// TwinCAT 3 PLC project plc_project
// ProgramVersion: 3.1.4022.1
// libraries:
//   Tc2_Standard, * (Beckhoff Automation GmbH)
//   Tc2_System, * (Beckhoff Automation GmbH)
//   Tc3_Module, * (Beckhoff Automation GmbH)
//   VisuDialogs, * (System)
//   VisuSymbols,3.5.10.0,System
// project tree:
//   / GlobalTextList.TcGTLO, PlcTask.TcTTO, Visualization Manager.TcVMO (not stored)
//   POUs/ MAIN.TcPOU, POU.TcPOU
//   VISUs/ Visualization.TcVIS

CONFIGURATION plc_project
    RESOURCE PLC ON TwinCAT3
        TASK PlcTask(INTERVAL := T#10ms, PRIORITY := 20);
        PROGRAM MAIN WITH PlcTask : MAIN;
    END_RESOURCE
END_CONFIGURATION

// ---- POUs/MAIN.TcPOU
PROGRAM MAIN
VAR
END_VAR

POU();

END_PROGRAM

// ---- POUs/POU.TcPOU
PROGRAM POU
VAR
	A: BOOL;
	B: BOOL;
	C: BOOL:= FALSE;
	add_result: UINT;
	sub_result: INT;
	mul_result: REAL;
	div_result: REAL;
	TON_0: TON;
	ton0_et: TIME;
	TOF_0: TOF;
	tof0_et: TIME;
	TP_0: TP;
	tp0_et: TIME;
	D: BOOL;
	CTD_0: CTD;
	CTD_1: CTD;
	ctd1_cv: WORD;
	Zero: BOOL;
	CTU_0: CTU;
	ctu0_cv: WORD;
	Maximum: BOOL;
END_VAR

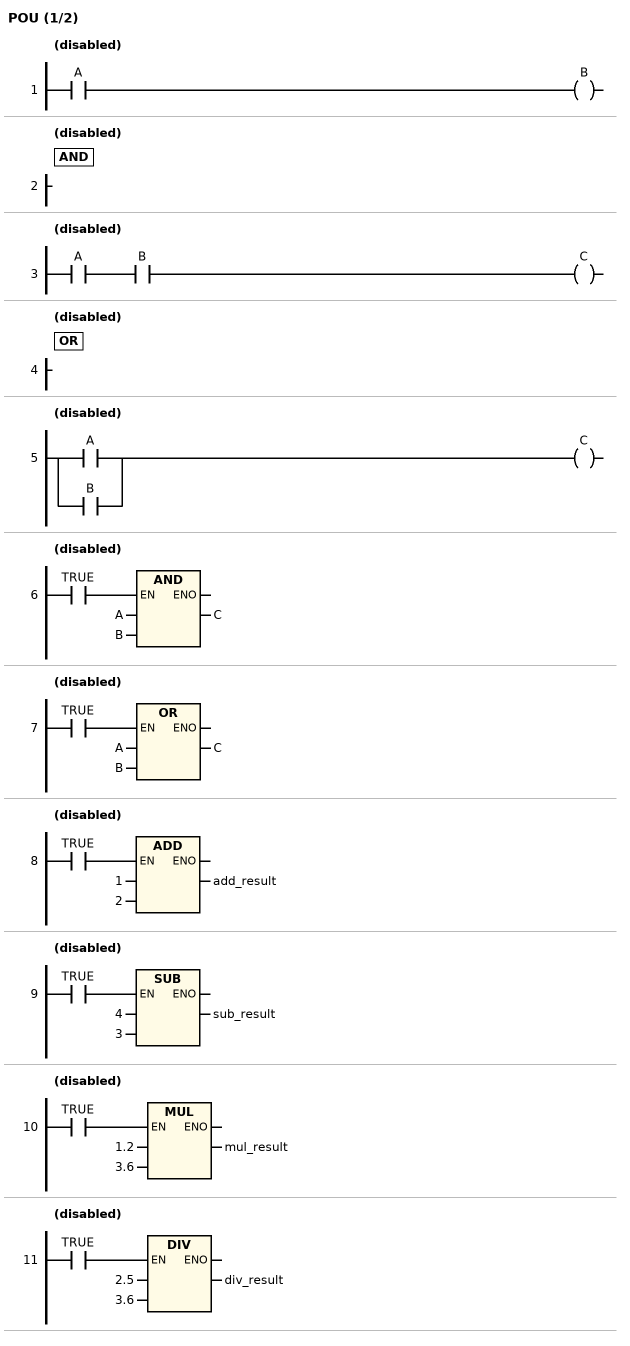
// NETWORK 1 (disabled)
// B := A;

// NETWORK 2 (disabled)
// label: AND

// NETWORK 3 (disabled)
// C := A AND B;

// NETWORK 4 (disabled)
// label: OR

// NETWORK 5 (disabled)
// C := A OR B;

// NETWORK 6 (disabled)
// C := A AND B;

// NETWORK 7 (disabled)
// C := A OR B;

// NETWORK 8 (disabled)
// add_result := 1 + 2;

// NETWORK 9 (disabled)
// sub_result := 4 - 3;

// NETWORK 10 (disabled)
// mul_result := 1.2 * 3.6;

// NETWORK 11 (disabled)
// div_result := 2.5 / 3.6;

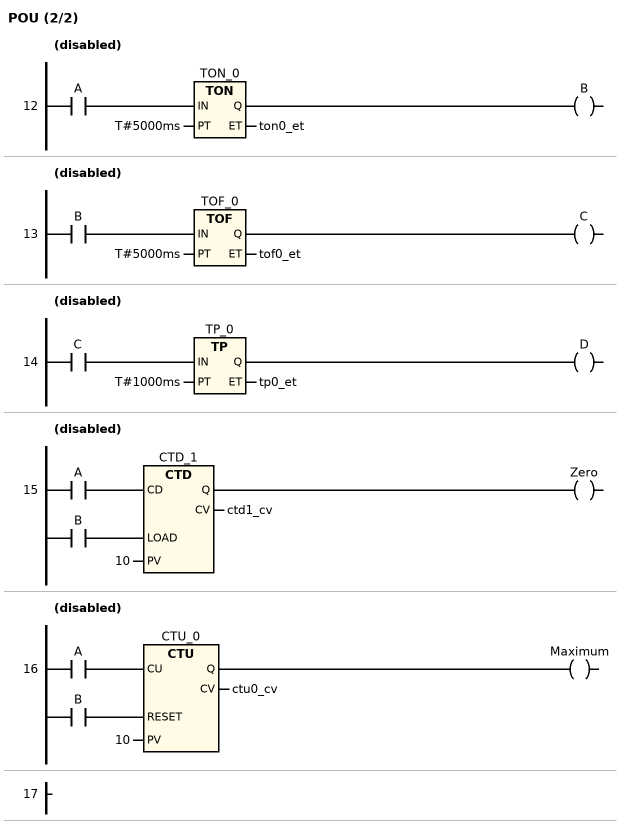
// NETWORK 12 (disabled)
// TON_0(IN := A, PT := T#5000ms, ET => ton0_et); // TON
// B := TON_0.Q;

// NETWORK 13 (disabled)
// TOF_0(IN := B, PT := T#5000ms, ET => tof0_et); // TOF
// C := TOF_0.Q;

// NETWORK 14 (disabled)
// TP_0(IN := C, PT := T#1000ms, ET => tp0_et); // TP
// D := TP_0.Q;

// NETWORK 15 (disabled)
// CTD_1(CD := A, LOAD := B, PV := 10, CV => ctd1_cv); // CTD
// Zero := CTD_1.Q;

// NETWORK 16 (disabled)
// CTU_0(CU := A, RESET := B, PV := 10, CV => ctu0_cv); // CTU
// Maximum := CTU_0.Q;

// NETWORK 17

END_PROGRAM

// ---- GlobalTextList.TcGTLO
TEXTLIST GlobalTextList
  495 = 'Button A'
  468 = 'LED A'
  950 = 'LED B'
  132 = 'LED C'
END_TEXTLIST

// ---- VISUs/Visualization.TcVIS
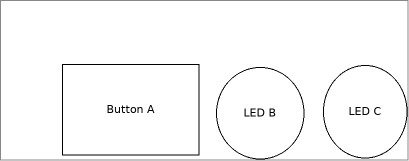
VISUALIZATION Visualization  // 409x161
    Rectangle (62,64 137x91), "Button A"
        OnMouseDown: toggle POU.A
    Ellipse (216,67 88x92), "LED B", colour toggle: POU.B
    Ellipse (323,65 84x93), "LED C", colour toggle: POU.C
END_VISUALIZATION
